// TIA Portal V19 export
FUNCTION "Rollformer_CALL" : Void   // FC162, LAD
TITLE = ROLLFORMER CALL
// stored: SetENOAutomatically false
   VAR_TEMP
      MissIO : Bool;
   END_VAR
BEGIN

REGION Network 1: Data In - PB Feed
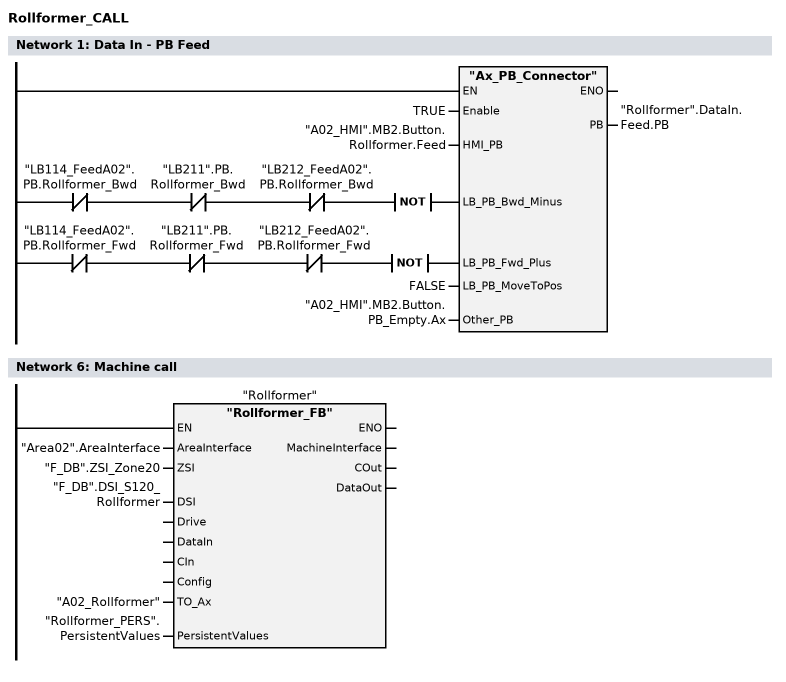
   RUNG wire#powerrail
      "Ax_PB_Connector"(LB_PB_Bwd_Minus := wire#w1, LB_PB_Fwd_Plus := wire#w2, Enable := TRUE, HMI_PB := "A02_HMI".MB2.Button.Rollformer.Feed, LB_PB_MoveToPos := FALSE, Other_PB := "A02_HMI".MB2.Button.PB_Empty.Ax, PB => "Rollformer".DataIn.Feed.PB)
   END_RUNG
   RUNG wire#powerrail
      I_Contact( "LB114_FeedA02".PB.Rollformer_Bwd )
      I_Contact( "LB211".PB.Rollformer_Bwd )
      I_Contact( "LB212_FeedA02".PB.Rollformer_Bwd )
      Not()
   END_RUNG wire#w1
   RUNG wire#powerrail
      I_Contact( "LB114_FeedA02".PB.Rollformer_Fwd )
      I_Contact( "LB211".PB.Rollformer_Fwd )
      I_Contact( "LB212_FeedA02".PB.Rollformer_Fwd )
      Not()
   END_RUNG wire#w2
   // the same network as SCL:
   "Ax_PB_Connector"(Enable := TRUE,
                     HMI_PB := "A02_HMI".MB2.Button.Rollformer.Feed,
                     LB_PB_Bwd_Minus := NOT (NOT "LB114_FeedA02".PB.Rollformer_Bwd AND NOT "LB211".PB.Rollformer_Bwd AND NOT "LB212_FeedA02".PB.Rollformer_Bwd),
                     LB_PB_Fwd_Plus := NOT (NOT "LB114_FeedA02".PB.Rollformer_Fwd AND NOT "LB211".PB.Rollformer_Fwd AND NOT "LB212_FeedA02".PB.Rollformer_Fwd),
                     LB_PB_MoveToPos := FALSE,
                     Other_PB := "A02_HMI".MB2.Button.PB_Empty.Ax,
                     PB => "Rollformer".DataIn.Feed.PB);
END_REGION

REGION Network 2 (SCL): DataIn - Sensor
   "Rollformer".DataIn.ConnectorPlugged1 := "A0201_Motore_Bancalata_1_Controllo_Connettore";
   "Rollformer".DataIn.ConnectorPlugged2 := "A0201_Motore_Bancalata_2_Controllo_Connettore";
   "Rollformer".DataIn.ConnectorPlugged3Side1 := "A0201_Motore_Bancalata_3_Lato_1_Controllo_Connettore";
   "Rollformer".DataIn.ConnectorPlugged3Side2 := "A0201_Motore_Bancalata_3_Lato_2_Controllo_Connettore";

   "Rollformer".DataIn.Feed.Fan_M_Feedback := "A0201_Ventilatore_Mot_Profila_Feedback";
END_REGION

REGION Network 3 (SCL): Drive

   "Rollformer".Drive.Infeed_ON := "Areas_ITF".AG.Infeed_Running;
   "Rollformer".Drive.AccessPoint := "HW_Const_Values".CU2_PN_585A1_ModuleAccessPoint;
   "Rollformer".Drive.AxisID := "CU2_ID_2_1190A1_1190M1";
   "Rollformer".Drive.TokenChain := "TOKENCHAIN_CU2";
END_REGION

REGION Network 4 (SCL): Config

   "Rollformer".Config.DataPresence := "PPrf_MAIN".ON_WORK.Header.PrgNo > 0;
   "Rollformer".Config.Data := "PPrf_MAIN".ON_WORK.A02_1_PartsCutting.Rollformer.TAxConfig;

   "Rollformer".Config.Feed := "A02_Config".Rollformer;
END_REGION

REGION Network 5 (SCL): CIn
   "Rollformer".CIn.ExtEnable_FlyingShareOk := "RollformingMng".FlyingCutoff.COut.Lead.LeadMovePermitted;
   "Rollformer".CIn.ExtEnable_MaterialCounterOK := NOT "PostPunchingMatCounter".COut.StopFeeding;
   "Rollformer".CIn.ExtEnable_MwFakCalcOk := NOT "MwFakCalc".COut.StopMaterialFeeding;
   "Rollformer".CIn.ExtEnable_UnloadRollwayOk := "AccRollConveyor".COut.Manager.RollformerFeedOk;

   "Rollformer".CIn.ExtEnable_LoopBwdOk := "Areas_ITF".A01.Loop1_COut.Exit_EnableFeedBkw;
   "Rollformer".CIn.ExtEnable_LoopFwdOk := "Areas_ITF".A01.Loop1_COut.Exit_EnableFeedFwd;
   "Rollformer".CIn.Loop1_VelOverride := "Areas_ITF".A01.Loop1_COut.Exit_VelocityOverride;

   "Rollformer".CIn.Manager := "RollformingMng".COut.Rollformer.Feed;

   "Rollformer".CIn.SOS_Enable := FALSE;
END_REGION

REGION Network 6: Machine call
   RUNG wire#powerrail
      "Rollformer"(AreaInterface := "Area02".AreaInterface, ZSI := "F_DB".ZSI_Zone20, DSI := "F_DB".DSI_S120_Rollformer, Drive :=, DataIn :=, CIn :=, Config :=, TO_Ax := "A02_Rollformer", PersistentValues := "Rollformer_PERS".PersistentValues, MachineInterface =>, COut =>, DataOut =>)
   END_RUNG
   // the same network as SCL:
   "Rollformer"(AreaInterface := "Area02".AreaInterface,   // "Rollformer_FB"
                ZSI := "F_DB".ZSI_Zone20,
                DSI := "F_DB".DSI_S120_Rollformer,
                TO_Ax := "A02_Rollformer",
                PersistentValues := "Rollformer_PERS".PersistentValues);
END_REGION

REGION Network 7 (SCL): Data Out
   "A0201_Ventilatore_Mot_Profila_Marcia" := "Rollformer".DataOut.Feed.Fan_M_Contactor;

   "A0201_Fine_Profila_V_Soffio_Pulizia_Phc_Tacca" := NOT "Rollformer".COut.Feed.Standstill;
END_REGION
END_FUNCTION
